(* CoDeSys 2.3.9.37 project: Cap3_3.pro *)
(* Libraries: Standard.LIB 4.10.05 12:14:46 *)

(* Global variable list: Global_Variables *)
VAR_GLOBAL

(* Variables de entrada *)
  P:BOOL;
  MI:BOOL;
  MD:BOOL;

(* Variables de salida *)
  KM1 : BOOL;
  KM2 : BOOL;

END_VAR

(* POU PLC_PRG, ST *)
PROGRAM PLC_PRG
VAR
  posy:INT;

END_VAR
Control();


IF KM1 THEN
  posy:=posy-1;
END_IF

IF KM2 THEN
  posy:=posy+1;
END_IF
END_PROGRAM

(* POU Control, LD *)
PROGRAM Control
VAR
END_VAR
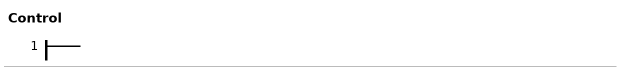
_LD_ (* Ladder Diagram *)
NETWORK 1
	*
_END_LD_
(* the same logic as Structured Text *)
(* Network 1 *)
END_PROGRAM

(* Visualisation Deposito
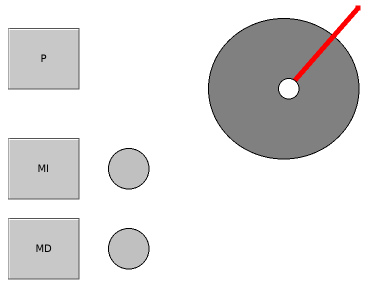
button at (50,80)-(121,141): text "P"; taps .P
button at (50,190)-(121,251): text "MI"; taps .MI
button at (50,270)-(121,331): text "MD"; taps .MD
polyline at (330,60)-(400,140): angle PLC_PRG.posy
ellipse at (150,200)-(191,241): alarm colour if .KM1
ellipse at (150,280)-(191,321): alarm colour if .KM2
2 more shapes without text or variables
*)
